// TIA Portal V17 export
// export: Created 2025-03-10T12:17:48.2062174Z, ExportSetting WithDefaults, DisplayName Totally Integrated Automation Portal, DisplayVersion V17 Update 8, DisplayName TIA Portal Openness, DisplayVersion V17 Update 8, DisplayName TIA Portal Version Control Interface, DisplayVersion V17, DisplayName SINAMICS Startdrive Advanced, DisplayVersion V17 SP2, DisplayName SINAMICS Startdrive G110M, G120, G120C, G120D, G120P, G115D, DisplayVersion V17 SP2, DisplayName SINAMICS Startdrive G130, G150, S120, S150, SINAMICS MV, S210, DisplayVersion V17 SP2, DisplayName STEP 7 Professional, DisplayVersion V17 Update 8, DisplayName SINUMERIK ONE STEP 7 Toolbox, DisplayVersion V17 Update 12, DisplayName SINUMERIK 840D sl STEP 7 Toolbox, DisplayVersion V17 Update 12, DisplayName STEP 7 Safety, DisplayVersion V17 Update 6, DisplayName WinCC Advanced, DisplayVersion V17 Update 8
TYPE "LBP_typeNCVariableToken"
TITLE = LBP_ReadVar and LBP_WriteVar Input Interface / Interfaz de entrada LBP_ReadVar y LBP_WriteVar / LBP_ReadVar und LBP_WriteVar Input Schnittstelle
// User Data Type for LBP_ReadVar[FB2] and LBP_WriteVar[FB3] Input Parameter Addrx / Tipo de datos de usuario para parámetros de entrada Addrx LBP_ReadVar[FB2] y LBP_WriteVar[FB3] / Anwenderdatentyp für LBP_ReadVar[FB2] und LBP_WriteVar[FB3] Eingangsparameter Addrx
// stored: IsFailsafeCompliant false
   STRUCT
      syntaxId : Byte;   // Syntaxkennung / syntax ID / ID de sintaxis
      areaAndUnit : Byte;   // Bereich und Einheit / area and unit / Área y unidad
      column : Word;   // Spalte / column / Columna
      row : Word;   // Zeile / row / Fila
      blockType : Byte;   // Blocktyp / block type / Tipo de bloque
      numberOfRows : Byte;   // Zeilenanzahl / number of rows / Número de filas
      dataTypeCode : Byte;   // Datentypcode / data type code / Código de tipo de datos
      length : Byte;   // Länge des Datentyps / length of data type / Longitud del tipo de datos
   END_STRUCT;
END_TYPE
